FUNCTION_BLOCK FB_Filler IMPLEMENTS IStation
VAR_INPUT
END_VAR
VAR_OUTPUT
END_VAR
VAR
	bPartPresent				: BOOL;
	bReady						: BOOL;
	bBusy						: BOOL;
	
	StationState				: E_StationState;
	pPartStatus					: POINTER TO ST_PartStatus;
	
	tmrWork						: TON;
	tmrDelay					: TON;
END_VAR

PROPERTY Busy : BOOL
GET
END_GET
END_PROPERTY

METHOD Execute : PVOID
VAR
	
END_VAR
CASE StationState OF
	
	E_StationState.IDLE:
		
		IF bPartPresent THEN
			tmrDelay(IN:=TRUE, PT:=T#500MS);
			IF tmrDelay.Q THEN
				StationState := E_StationState.WORKING;
			END_IF
		ELSE
			bReady := TRUE;
			bBusy := FALSE;
		END_IF
		
	E_StationState.WORKING:
		
		bReady := FALSE;
		bBusy := TRUE;
		
		tmrWork(IN:= TRUE, PT:=T#1.5S);
		IF tmrWork.Q THEN
			StationState := E_StationState.DONE;
			tmrWork(IN:=FALSE);
		END_IF
	
	E_StationState.DONE:
	
		bReady := TRUE;
		bBusy := FALSE;
		
		IF NOT bPartPresent THEN
			IF PartStatus <> 0 THEN
				PartStatus^.bFillerStatus := TRUE;
			END_IF
			StationState := E_StationState.IDLE;
		END_IF
		
END_CASE
END_METHOD

PROPERTY Faulted : BOOL
GET
END_GET
END_PROPERTY

PROPERTY PartPresent : BOOL
GET
PartPresent := bPartPresent;
END_GET
END_PROPERTY

PROPERTY PartStatus : POINTER TO ST_PartStatus
GET
END_GET
SET
END_SET
END_PROPERTY

PROPERTY Ready : BOOL
GET
Ready := bReady;
END_GET
END_PROPERTY

END_FUNCTION_BLOCK

(* stored: Version 1.1.0.1, ProductVersion 3.1.4024.12
   POU FB_Filler: Id {6295f515-0cbf-4a9e-9a05-3f3e3f3d6db2}, SpecialFunc None
   Property Busy: Id {7b22d881-ebdb-4f3f-befe-dc51dc54aaa2}
   Get Get: Id {ca417ef2-f1af-4039-b554-114d2928bdf1}
   Method Execute: Id {ff5674ff-bdfb-419d-a54e-f90304492f60}
   Property Faulted: Id {2979689c-56ae-45ad-889c-8947b962ccd6}
   Get Get: Id {ac2e006c-b510-42e2-8be1-91884283522f}
   Property PartPresent: Id {95bfdd99-c2ff-4ea8-a069-a6af56c1f591}
   Get Get: Id {c1570d8d-2d16-4701-b97f-5e49092a4e7e}
   Property PartStatus: Id {cfb0896c-0015-4e79-83bb-e427abd35db0}
   Get Get: Id {4dd7c970-06df-4ded-8394-62151b37c1ec}
   Set Set: Id {caafe008-208b-409e-8c59-94a3eb8658cc}
   Property Ready: Id {0c567ab7-f2cc-4ae2-bbee-7022ed467954}
   Get Get: Id {c6abe93d-9dd7-495c-9228-987f2d612abd} *)
